PROGRAM MAIN
VAR

END_VAR

single.checkPower();
single.checkMoving();
single.checkRelMove();
single.checkHalt();
single.checkStop();
single.checkReset();
single.checkAdjustingVelocity();
single.checkSetPoint();
single.checkGoHome();

END_PROGRAM

(* stored: Version 1.1.0.1, ProductVersion 3.1.4024.4
   POU MAIN: Id {17d55ee0-0987-40b0-829c-2cffe93b08a6}, SpecialFunc None *)
